FUNCTION_BLOCK "funcB1"
{ S7_Optimized_Access := 'TRUE' }
VERSION : 0.1

BEGIN
	//some code
	//
	//
END_FUNCTION_BLOCK

